Staubli VAL3: getLastId.pgx

public program getLastId(num& x_nMoveId)
begin
  // give back the last ID
  x_nMoveId=aAction[size(aAction)-1].nMoveId
end
